// TIA Portal V19 export
DATA_BLOCK "A0302_HU_Cytropack"   // DB81
// stored: InstanceOfName A0302_HU_Cytropack_FB, InstanceOfType FB
"A0302_HU_Cytropack_FB"
   // VAR_INPUT
   //    AreaInterface : "AreaInterface";
   //    ZSI : "udt_ZoneSafetyInterface";
   //    DSI : "udt_DeviceSafetyInterface";
   //    DataIn : Struct
   //       Pb_Stop : Bool;
   //       Pb_Start : Bool;
   //    END_STRUCT;
   //    CIn : Struct
   //       Manager : Struct
   //          EnableStopDoorOpeningReq { ExternalWritable := 'False'} : Bool;
   //          EnableStopInPhase { ExternalWritable := 'False'} : Bool;
   //          EnableStopProgrammed { ExternalWritable := 'False'} : Bool;
   //          Control_ON { ExternalWritable := 'False'} : Bool;
   //          Rest { ExternalWritable := 'False'} : Bool;
   //          Work { ExternalWritable := 'False'} : Bool;
   //       END_STRUCT;
   //       SemiAut_Pb { ExternalAccessible := 'False'; ExternalVisible := 'False'; ExternalWritable := 'False'} : Bool;
   //       PressureReq : Bool;
   //       PressureRunning : Bool;
   //       CarroPareggTesta : Struct
   //          Bloccaggio { ExternalAccessible := 'False'; ExternalVisible := 'False'; ExternalWritable := 'False'} : "ValveMachine_COut";
   //       END_STRUCT;
   //       CarroPareggCoda : Struct
   //          Bloccaggio { ExternalAccessible := 'False'; ExternalVisible := 'False'; ExternalWritable := 'False'} : "ValveMachine_COut";
   //          PareggiatoreLong { ExternalAccessible := 'False'; ExternalVisible := 'False'; ExternalWritable := 'False'} : "ValveMachine_COut";
   //       END_STRUCT;
   //    END_STRUCT;
   //    InputADDR : HW_IO;
   //    OutputADDR : HW_IO;
   // END_VAR
   // VAR_OUTPUT
   //    MachineInterface : "MachineInterface";
   //    COut : Struct
   //       Standstill : Bool;
   //       Run_CheckNext : Bool;
   //       CtrlSafe : Bool;
   //       PressureRunning : Bool;
   //       PressureInTarget : Bool;
   //    END_STRUCT;
   // END_VAR
   // VAR_IN_OUT
   //    Par : Struct
   //       Bloccaggio : Struct
   //          TargetPressure : Real;
   //          TargetSpeed : Real;
   //          Delta : Struct
   //             Min : Real;
   //             Max : Real;
   //          END_STRUCT;
   //       END_STRUCT;
   //       Pareggiamento : Struct
   //          TargetPressure : Real;
   //          TargetSpeed : Real;
   //          Delta : Struct
   //             Min : Real;
   //             Max : Real;
   //          END_STRUCT;
   //       END_STRUCT;
   //    END_STRUCT;
   // END_VAR
   // VAR
   //    M_Chiller : "Motor";
   //    Sts : Struct
   //       Standstill : Bool;
   //       AlarmsPresence : Bool;
   //       WarningsPresence : Bool;
   //       Cnd : Bool;
   //    END_STRUCT;
   //    Ctrl : Struct
   //       StopDueDoorOpeningRequest : Bool;
   //       StopInPhase : Bool;
   //       StopProgrammed : Bool;
   //       StopAborting : Bool;
   //       Run : Bool;
   //       Run_Man : Bool;
   //       Run_Aut : Bool;
   //    END_STRUCT;
   //    Alarm : Struct
   //       M_Chiller { S7_SetPoint := 'True'} : "MotorAlr";
   //       Fc_P5020 : Struct
   //          Error { S7_SetPoint := 'True'} : Bool;
   //          Warning : Bool;
   //       END_STRUCT;
   //       Fc_Diagn : Struct
   //          "0" : Bool;
   //          "1" : Bool;
   //          "2" : Bool;
   //          "3" : Bool;
   //          "4" : Bool;
   //          "5" : Bool;
   //          "6" : Bool;
   //          "7" : Bool;
   //          "8" : Bool;
   //          "9" : Bool;
   //          "10" : Bool;
   //          "11" : Bool;
   //          "12" : Bool;
   //          "13" : Bool;
   //          "14" : Bool;
   //          "15" : Bool;
   //       END_STRUCT;
   //    END_STRUCT;
   //    Warning : Struct
   //       NotAutReady : Bool;
   //    END_STRUCT;
   //    TON_NoPendingCmd : IEC_TIMER;
   //    TON_Inactivity : IEC_TIMER;
   //    TON_Pressure { S7_SetPoint := 'True'} : IEC_TIMER;
   //    Aux : Struct
   //       Pb_Start : Bool;
   //       ReqParBloccaggio : Bool;
   //       ReqParParegg : Bool;
   //    END_STRUCT;
   //    iReturnVal : Int;
   //    Error : Bool;
   //    bFBErrorDPRD_DPWR : Bool;
   //    stInputData { S7_SetPoint := 'True'} : "FCP_IN";
   //    stOutputData { S7_SetPoint := 'True'} : "FCP_OUT";
   //    Range_TargetBlocc : Struct
   //       Min : Real;
   //       Max : Real;
   //    END_STRUCT;
   //    Range_TargetParegg : Struct
   //       Min : Real;
   //       Max : Real;
   //    END_STRUCT;
   //    Target : Struct
   //       Pressure_Value { ExternalAccessible := 'False'; ExternalVisible := 'False'; ExternalWritable := 'False'} : Real;
   //       MaxSpeed_Value { ExternalAccessible := 'False'; ExternalVisible := 'False'; ExternalWritable := 'False'} : Real;
   //    END_STRUCT;
   // END_VAR
BEGIN
END_DATA_BLOCK
